INTERFACE I_NciCommand EXTENDS I_Command

END_INTERFACE

(* stored: Version 1.1.0.1, ProductVersion 3.1.4024.12
   Itf I_NciCommand: Id {31172878-ef3e-095d-0185-2a29859dec6d} *)
